(* CODESYS project Automation.library
   Company: Ziga Javornik
   DefaultNamespace: ZigaLibs.Automation
   Version: 0.0.1.2
   Placeholder: ZigaLibs.Automation
   Author: Ziga Javornik
   Description: Function blocks used for general automation.
   Title: ZigaLibs.Automation

Project tree, tasks and I/O mapping:
  libraries: Tc2_Standard, * (Beckhoff Automation GmbH); Tc2_System, * (Beckhoff Automation GmbH); Tc3_Module, * (Beckhoff Automation GmbH); TcUnit, * (www.tcunit.org); ZigaLibs.ProcessControl, 0.0.2.3 (Ziga Javornik); ZigaLibs.Core, 0.0.3.7 (Ziga Javornik)
  GVLs/
  SOURCE/
    FrequencyInverter/
      data type E_FqInverterState
      function block FB_FqInverter [ST]: CalculateFeedback, CalculateSetpoint, Enabled, Error, FB_init, Frequency, MaxFrequency, Reset, SetpointDeviation
      function block FB_FqInverter_IO [ST]: CalculateFeedback, CalculateSetpoint, Enabled, Error, FB_init, Frequency, MaxFrequency, Reset, SetpointDeviation
      interface I_FqInverter: Enabled, Error, Frequency, MaxFrequency, Reset
      data type ST_FqInverter_HwInputs
      data type ST_FqInverter_HwOutputs
    LightTower/
      function block FB_LightTower [ST]: Buzzer, FB_init, GreenLight, OrangeLight, RedLight
      function block FB_LightTowerComponent [ST]: Activate, Deactivate, FB_init, PulseWithInterval, Value
      interface I_LightTower: Buzzer, GreenLight, OrangeLight, RedLight
      interface I_LightTowerComponent: Activate, Deactivate, PulseWithInterval, Value
    MFC/
      data type ST_MfcCommands
      data type ST_MfcFeedback
  TESTS/
    Test suites/
      function block FB_FqInverter_IO_Tests [ST]: Test01_WhenDisabledOutputIsAlwaysFalse, Test02_Enable_ExpectOutputAccordingToMaxFrequencySetting, Test03_SetNegativeMaximumFrequency_ExpectOutputAlways0, Test04_SetNegativeSetpoint_ExpectOutputAlways0, Test05_DeviationIsOnlyActiveWhenEnabled, Test06_InverterErrorActive_ExpectOutputAlways0, Test07_Reset_ExpectPulseOnOutput_WhenNoErrorExpectNothing, TestXX_Template
      function block FB_LightTower_Tests [ST]: Test01_GreenLight_ActivateDeactivate_VerifyReferencedVariableValue, Test02_OrangeLight_ActivateDeactivate_VerifyReferencedVariableValue, Test03_RedLight_ActivateDeactivate_VerifyReferencedVariableValue, Test04_Buzzer_ActivateDeactivate_VerifyReferencedVariableValue
      function block FB_LightTowerComponent_Tests [ST]: Test01_AllFunctionalityTests
    program PRG_TESTS [ST]
*)

// SOURCE/FrequencyInverter/E_FqInverterState
{attribute 'qualified_only'}
{attribute 'strict'}
TYPE E_FqInverterState :
(
	DISABLED,
	ENABLED,
	RUNNING,
	ERROR,
	RESET
);
END_TYPE

// SOURCE/FrequencyInverter/ST_FqInverter_HwInputs
TYPE ST_FqInverter_HwInputs :
STRUCT
	Feedback	: INT;	// Actual feedback value
	Error		: BOOL;	// Error indication
	Ready		: BOOL;	// Ready indication
END_STRUCT
END_TYPE

// SOURCE/FrequencyInverter/ST_FqInverter_HwOutputs
TYPE ST_FqInverter_HwOutputs :
STRUCT
	Setpoint	: INT;	// Setpoint value
	Enable		: BOOL;	// Enable operation
	Reset		: BOOL;	// Reset error
END_STRUCT
END_TYPE

// SOURCE/MFC/ST_MfcCommands
TYPE ST_MfcCommands :
STRUCT
	FlowSetpoint	: REAL;
	Enable			: BOOL;
END_STRUCT
END_TYPE

// SOURCE/MFC/ST_MfcFeedback
TYPE ST_MfcFeedback :
STRUCT
	ValvePosition	: REAL;
	ActualFlow		: REAL;
END_STRUCT
END_TYPE

// SOURCE/FrequencyInverter/FB_FqInverter
// A simple frequency invert trough IO signals function block. 
// The difference to FB_FqInverter_IO is that this block uses reference assignment instead of having IO signals generated trough process image
// Constructor parameters:
(*
	(setpointMaximumValue	:= 32767,	//INT; Maximum setpoint value, ging to terminal   
	feedbackMaximumValue	:= 32767,	//INT; Maximum feedback value coming from terminal
	maximumFrequency		:= 50.0,	//REAL; Maximum frequency
	// Output signals, going to inverter
	enableSignal	:= , // REFERENCE TO BOOL;
	resetSignal		:= , // REFERENCE TO BOOL;
	setpointSignal	:= , // REFERENCE TO INT;
	// Input signals, coming from inverter
	errorSignal		:= , // REFERENCE TO BOOL;
	feedbackSignal	:= ); // REFERENCE TO INT;
*)
FUNCTION_BLOCK FB_FqInverter IMPLEMENTS I_FqInverter
VAR
	_enabled				: BOOL;
	_error					: BOOL;
	_frequency				: ZigaLibs_Core.ST_Value;
	_maxFrequency			: REAL;
	_state					: E_FqInverterState;
	_setpointMaximumValue	: INT;
	_feedbackMaximumValue	: INT;
	_setpointDeviation			: ZigaLibs_ProcessControl.FB_ValueDeviation;
	
	// Output signals, going to inverter
	_enableSignal	: REFERENCE TO BOOL;
	_resetSignal	: REFERENCE TO BOOL;
	_setpointSignal	: REFERENCE TO INT;
	// Input signals, coming from inverter
	_errorSignal	: REFERENCE TO BOOL;
	_feedbackSignal	: REFERENCE TO INT;
END_VAR

_frequency.Actual := CalculateFeedback();

IF _errorSignal AND _state <> E_FqInverterState.RESET THEN
	_State := E_FqInverterState.ERROR;
END_IF


CASE _state OF
	E_FqInverterState.DISABLED:
		_enableSignal := FALSE;
		_setpointSignal := 0;
		IF _enabled THEN
			_state := E_FqInverterState.ENABLED;
		END_IF
		
	E_FqInverterState.ENABLED:
		IF NOT _enabled THEN
			_state := E_FqInverterState.DISABLED;
		ELSE
			_enableSignal := TRUE;
			_setpointSignal := CalculateSetpoint();
		END_IF
		
	E_FqInverterState.ERROR:
		_error := TRUE;
		_enableSignal := FALSE;
		_setpointSignal := 0;
		
	E_FqInverterState.RESET:
		_error := FALSE;
		_enableSignal := FALSE;
		_setpointSignal := 0;
		_resetSignal := FALSE;
		IF NOT _errorSignal THEN
			_state := E_FqInverterState.DISABLED;
		END_IF
END_CASE

_setpointDeviation.Enable := _state = E_FqInverterState.ENABLED;
_setpointDeviation.Value.Actual := _frequency.Actual;
_setpointDeviation.Value.Setpoint := _frequency.Setpoint;
_setpointDeviation();

METHOD PRIVATE CalculateFeedback : REAL
VAR_INPUT
END_VAR
// Invalid parameter setting.
IF _feedbackMaximumValue <= 0 OR _maxFrequency < 0 THEN
	CalculateFeedback := 0;
ELSE
	CalculateFeedback := _maxFrequency * (INT_TO_REAL(_feedbackSignal) / INT_TO_REAL(_feedbackMaximumValue));
END_IF
END_METHOD

METHOD PRIVATE CalculateSetpoint : INT
VAR_INPUT
END_VAR
VAR
	validatedFrequencySetpoint	: REAL;
	frequencySetpointFraction	: REAL;
END_VAR
// Limit setpoint between 0 and max
validatedFrequencySetpoint := MAX(0, MIN(_maxFrequency, _frequency.Setpoint));

// If max frequency is 0, invalid setting
IF _maxFrequency <= 0 THEN
	frequencySetpointFraction := 0;
ELSE
	frequencySetpointFraction := validatedFrequencySetpoint / _maxFrequency;
END_IF

CalculateSetpoint := REAL_TO_INT(frequencySetpointFraction * _setpointMaximumValue);
END_METHOD

{attribute 'monitoring':='call'}
(* Gets or sets whether or not the unit is enabled.*)
PROPERTY Enabled : BOOL
GET
Enabled := _enabled;
END_GET
SET
_enabled := Enabled;
END_SET
END_PROPERTY

{attribute 'monitoring':='call'}
(* Returns TRUE if an error is active*)
PROPERTY Error : BOOL
GET
Error := _error;
END_GET
END_PROPERTY

METHOD FB_init : BOOL
VAR_INPUT
	bInitRetains : BOOL; // if TRUE, the retain variables are initialized (warm start / cold start)
	bInCopyCode : BOOL;  // if TRUE, the instance afterwards gets moved into the copy code (online change)
	setpointMaximumValue	: INT;	// Maximum setpoint value, ging to terminal
	feedbackMaximumValue	: INT;	// Maximum feedback value coming from terminal
	maximumFrequency		: REAL;	// Maximum frequency
	// Output signals, going to inverter
	enableSignal	: REFERENCE TO BOOL;
	resetSignal		: REFERENCE TO BOOL;
	setpointSignal	: REFERENCE TO INT;
	// Input signals, coming from inverter
	errorSignal		: REFERENCE TO BOOL;
	feedbackSignal	: REFERENCE TO INT;
END_VAR
_setpointMaximumValue := setpointMaximumValue;
_feedbackMaximumValue := feedbackMaximumValue;
_maxFrequency := maximumFrequency;
_enableSignal REF= enableSignal;
_resetSignal REF= resetSignal;
_setpointSignal REF= setpointSignal;
_errorSignal REF= errorSignal;
_feedbackSignal REF= feedbackSignal;
END_METHOD

{attribute 'monitoring':='call'}
(* Provides access to frequncy setpoint and actual value*)
PROPERTY Frequency : REFERENCE TO ZigaLibs_Core.ST_Value
GET
Frequency REF= _frequency;
END_GET
SET
_frequency := Frequency;
END_SET
END_PROPERTY

{attribute 'monitoring':='call'}
(* Gets or sets the maximum frequency.*)
PROPERTY MaxFrequency : REAL
GET
MaxFrequency := _maxFrequency;
END_GET
SET
_maxFrequency := MaxFrequency;
END_SET
END_PROPERTY

(* If an error is active, it will be reset.*)
METHOD Reset
VAR_INST
	resetTimer	: Tc2_Standard.TON := (PT := T#200MS);
END_VAR
IF _errorSignal THEN
	resetTimer(IN := NOT resetTimer.Q, PT := T#100MS);
	_resetSignal := NOT resetTimer.Q;
ELSE
	resetTimer(IN := FALSE);
	_resetSignal := FALSE;
	_state := E_FqInverterState.RESET;
END_IF
END_METHOD

{attribute 'monitoring':='call'}
PROPERTY SetpointDeviation : ZigaLibs_ProcessControl.I_ValueDeviationLimited
GET
SetpointDeviation := _setpointDeviation;
END_GET
END_PROPERTY

END_FUNCTION_BLOCK

// SOURCE/FrequencyInverter/FB_FqInverter_IO
// A simple frequency invert trough IO signals function block
// Constructor parameters:
(*
	(setpointMaximumValue	:= 32767,	//INT; Maximum setpoint value, ging to terminal   
	feedbackMaximumValue	:= 32767,	//INT; Maximum feedback value coming from terminal
	maximumFrequency		:= 50.0);	//REAL; Maximum frequency                         

*)
FUNCTION_BLOCK FB_FqInverter_IO IMPLEMENTS I_FqInverter
VAR
	_enabled				: BOOL;
	_error					: BOOL;
	_frequency				: ZigaLibs_Core.ST_Value;
	_maxFrequency			: REAL;
	_state					: E_FqInverterState;
	_setpointMaximumValue	: INT;
	_feedbackMaximumValue	: INT;
	_setpointDeviation			: ZigaLibs_ProcessControl.FB_ValueDeviation;
END_VAR

VAR
	Inputs	AT %I* 	: ST_FqInverter_HwInputs;
	Outputs	AT %Q*	: ST_FqInverter_HwOutputs;
END_VAR

_frequency.Actual := CalculateFeedback();

IF Inputs.Error AND _state <> E_FqInverterState.RESET THEN
	_State := E_FqInverterState.ERROR;
END_IF


CASE _state OF
	E_FqInverterState.DISABLED:
		Outputs.Enable := FALSE;
		Outputs.Setpoint := 0;
		IF _enabled THEN
			_state := E_FqInverterState.ENABLED;
		END_IF
		
	E_FqInverterState.ENABLED:
		IF NOT _enabled THEN
			_state := E_FqInverterState.DISABLED;
		ELSE
			Outputs.Enable := TRUE;
			Outputs.Setpoint := CalculateSetpoint();
		END_IF
		
	E_FqInverterState.ERROR:
		_error := TRUE;
		Outputs.Enable := FALSE;
		Outputs.Setpoint := 0;
		
	E_FqInverterState.RESET:
		_error := FALSE;
		Outputs.Enable := FALSE;
		Outputs.Setpoint := 0;
		outputs.Reset := FALSE;
		IF NOT Inputs.Error THEN
			_state := E_FqInverterState.DISABLED;
		END_IF
END_CASE

_setpointDeviation.Enable := _state = E_FqInverterState.ENABLED;
_setpointDeviation.Value.Actual := _frequency.Actual;
_setpointDeviation.Value.Setpoint := _frequency.Setpoint;
_setpointDeviation();

METHOD PRIVATE CalculateFeedback : REAL
VAR_INPUT
END_VAR
// Invalid parameter setting.
IF _feedbackMaximumValue <= 0 OR _maxFrequency < 0 THEN
	CalculateFeedback := 0;
ELSE
	CalculateFeedback := _maxFrequency * (INT_TO_REAL(Inputs.Feedback) / INT_TO_REAL(_feedbackMaximumValue));
END_IF
END_METHOD

METHOD PRIVATE CalculateSetpoint : INT
VAR_INPUT
END_VAR
VAR
	validatedFrequencySetpoint	: REAL;
	frequencySetpointFraction	: REAL;
END_VAR
// Limit setpoint between 0 and max
validatedFrequencySetpoint := MAX(0, MIN(_maxFrequency, _frequency.Setpoint));

// If max frequency is 0, invalid setting
IF _maxFrequency <= 0 THEN
	frequencySetpointFraction := 0;
ELSE
	frequencySetpointFraction := validatedFrequencySetpoint / _maxFrequency;
END_IF

CalculateSetpoint := REAL_TO_INT(frequencySetpointFraction * _setpointMaximumValue);
END_METHOD

{attribute 'monitoring':='call'}
(* Gets or sets whether or not the unit is enabled.*)
PROPERTY Enabled : BOOL
GET
Enabled := _enabled;
END_GET
SET
_enabled := Enabled;
END_SET
END_PROPERTY

{attribute 'monitoring':='call'}
(* Returns TRUE if an error is active*)
PROPERTY Error : BOOL
GET
Error := _error;
END_GET
END_PROPERTY

METHOD FB_init : BOOL
VAR_INPUT
	bInitRetains : BOOL; // if TRUE, the retain variables are initialized (warm start / cold start)
	bInCopyCode : BOOL;  // if TRUE, the instance afterwards gets moved into the copy code (online change)
	setpointMaximumValue	: INT;	// Maximum setpoint value, ging to terminal
	feedbackMaximumValue	: INT;	// Maximum feedback value coming from terminal
	maximumFrequency		: REAL;	// Maximum frequency
END_VAR
_setpointMaximumValue := setpointMaximumValue;
_feedbackMaximumValue := feedbackMaximumValue;
_maxFrequency := maximumFrequency;
END_METHOD

{attribute 'monitoring':='call'}
(* Provides access to frequncy setpoint and actual value*)
PROPERTY Frequency : REFERENCE TO ZigaLibs_Core.ST_Value
GET
Frequency REF= _frequency;
END_GET
SET
_frequency := Frequency;
END_SET
END_PROPERTY

{attribute 'monitoring':='call'}
(* Gets or sets the maximum frequency.*)
PROPERTY MaxFrequency : REAL
GET
MaxFrequency := _maxFrequency;
END_GET
SET
_maxFrequency := MaxFrequency;
END_SET
END_PROPERTY

(* If an error is active, it will be reset.*)
METHOD Reset
VAR_INST
	resetTimer	: Tc2_Standard.TON := (PT := T#200MS);
END_VAR
IF Inputs.Error THEN
	resetTimer(IN := NOT resetTimer.Q, PT := T#100MS);
	Outputs.Reset := NOT resetTimer.Q;
ELSE
	resetTimer(IN := FALSE);
	Outputs.Reset := FALSE;
	_state := E_FqInverterState.RESET;
END_IF
END_METHOD

{attribute 'monitoring':='call'}
PROPERTY SetpointDeviation : ZigaLibs_ProcessControl.I_ValueDeviationLimited
GET
SetpointDeviation := _setpointDeviation;
END_GET
END_PROPERTY

END_FUNCTION_BLOCK

// SOURCE/FrequencyInverter/I_FqInverter
INTERFACE I_FqInverter

{attribute 'monitoring':='call'}
// Gets or sets whether or not the unit is enabled.
PROPERTY Enabled : BOOL
GET
END_GET
SET
END_SET
END_PROPERTY

{attribute 'monitoring':='call'}
// Returns TRUE if an error is active
PROPERTY Error : BOOL
GET
END_GET
END_PROPERTY

{attribute 'monitoring':='call'}
// Provides access to frequncy setpoint and actual value
PROPERTY Frequency : REFERENCE TO ZigaLibs_Core.ST_Value
GET
END_GET
SET
END_SET
END_PROPERTY

{attribute 'monitoring':='call'}
// Gets or sets the maximum frequency.
PROPERTY MaxFrequency : REAL
GET
END_GET
SET
END_SET
END_PROPERTY

// If an error is active, it will be reset.
METHOD Reset
END_METHOD

END_INTERFACE

// SOURCE/LightTower/FB_LightTower
(* Provides acces to control the light tower components.
Constructor template as follows:
	(greenLight		:= ,// REFERENCE TO BOOL;
	orangeLight		:= ,// REFERENCE TO BOOL;
	redLight		:= ,// REFERENCE TO BOOL;
	buzzer			:= );// REFERENCE TO BOOL;
*)

FUNCTION_BLOCK FB_LightTower IMPLEMENTS I_LightTower
VAR	
	_redLightControl	: FB_LightTowerComponent;
	_orangeLightControl	: FB_LightTowerComponent;
	_greenLightControl	: FB_LightTowerComponent;
	_buzzerControl		: FB_LightTowerComponent;
END_VAR

_redLightControl();
_orangeLightControl();
_greenLightControl();
_buzzerControl();

// Provides access to buzzer control
PROPERTY Buzzer : I_LightTowerComponent
GET
Buzzer := _buzzerControl;
END_GET
END_PROPERTY

METHOD FB_init : BOOL
VAR_INPUT
	bInitRetains 	: BOOL; // if TRUE, the retain variables are initialized (warm start / cold start)
	bInCopyCode 	: BOOL;  // if TRUE, the instance afterwards gets moved into the copy code (online change)
	greenLight		: REFERENCE TO BOOL;
	orangeLight		: REFERENCE TO BOOL;
	redLight		: REFERENCE TO BOOL;
	buzzer			: REFERENCE TO BOOL;
END_VAR
_greenLightControl.component REF= greenLight;
_orangeLightControl.component REF= orangeLight;
_redLightControl.component REF= redLight;
_buzzerControl.component REF= buzzer;
END_METHOD

// Provides access to green light control
PROPERTY GreenLight : I_LightTowerComponent
GET
GreenLight := _greenLightControl;
END_GET
END_PROPERTY

// Provides access to orange light control
PROPERTY OrangeLight : I_LightTowerComponent
GET
OrangeLight := _orangeLightControl;
END_GET
END_PROPERTY

// Provides access to red light control
PROPERTY RedLight : I_LightTowerComponent
GET
RedLight := _redLightControl;
END_GET
END_PROPERTY

END_FUNCTION_BLOCK

// SOURCE/LightTower/I_LightTower
INTERFACE I_LightTower

// Provides access to buzzer control
PROPERTY Buzzer : I_LightTowerComponent
GET
END_GET
END_PROPERTY

// Provides access to green light control
PROPERTY GreenLight : I_LightTowerComponent
GET
END_GET
END_PROPERTY

// Provides access to orange light control
PROPERTY OrangeLight : I_LightTowerComponent
GET
END_GET
END_PROPERTY

// Provides access to red light control
PROPERTY RedLight : I_LightTowerComponent
GET
END_GET
END_PROPERTY

END_INTERFACE

// SOURCE/LightTower/I_LightTowerComponent
INTERFACE I_LightTowerComponent

// Sets the component state to TRUE.
METHOD Activate
VAR_INPUT
END_VAR
END_METHOD

// Sets the component state to FALSE.
METHOD Deactivate
VAR_INPUT
END_VAR
END_METHOD

METHOD PulseWithInterval
VAR_INPUT
	DurationOn	: TIME;
	DurationOff	: TIME;
END_VAR
END_METHOD

{attribute 'monitoring':='call'}
// Gets the current state of the component
PROPERTY Value : BOOL
GET
END_GET
END_PROPERTY

END_INTERFACE

// SOURCE/LightTower/FB_LightTowerComponent
FUNCTION_BLOCK FB_LightTowerComponent IMPLEMENTS I_LightTowerComponent
VAR_INPUT
	component : REFERENCE TO BOOL;
END_VAR
VAR
	_component	: ZigaLibs_Core.BoolEx := (variable := component);
END_VAR

_component(variable := component);

METHOD Activate
IF NOT __ISVALIDREF(component) THEN
	RETURN;
END_IF
_component.Set();
END_METHOD

METHOD Deactivate
IF NOT __ISVALIDREF(component) THEN
	RETURN;
END_IF
_component.Reset();
END_METHOD

METHOD FB_init : BOOL
VAR_INPUT
	bInitRetains : BOOL; // if TRUE, the retain variables are initialized (warm start / cold start)
	bInCopyCode : BOOL;  // if TRUE, the instance afterwards gets moved into the copy code (online change)
END_VAR
END_METHOD

METHOD PulseWithInterval
VAR_INPUT
	DurationOn	: TIME;
	DurationOff	: TIME;
END_VAR
VAR_INST
	timerOn		: Tc2_Standard.TON;
	timerOff	: Tc2_Standard.TON;
END_VAR
IF NOT __ISVALIDREF(component) THEN
	RETURN;
END_IF
_component.PulseWithInterval(DurationOn,DurationOff);
END_METHOD

{attribute 'monitoring':='call'}
(* Gets the current state of the component*)
PROPERTY Value : BOOL
GET
Value := _component.Value;
END_GET
END_PROPERTY

END_FUNCTION_BLOCK

// TESTS/Test suites/FB_FqInverter_IO_Tests
FUNCTION_BLOCK INTERNAL FB_FqInverter_IO_Tests EXTENDS FB_TestSuite
VAR_INPUT
END_VAR
VAR_OUTPUT
END_VAR
VAR
	_fqInvert : FB_FqInverter_IO(
		setpointMaximumValue	:= 32767,	//INT; Maximum setpoint value, ging to terminal   
		feedbackMaximumValue	:= 32767,	//INT; Maximum feedback value coming from terminal
		maximumFrequency		:= 50.0);	//REAL; Maximum frequency     
END_VAR

Test01_WhenDisabledOutputIsAlwaysFalse();
Test02_Enable_ExpectOutputAccordingToMaxFrequencySetting();
Test03_SetNegativeMaximumFrequency_ExpectOutputAlways0();
Test04_SetNegativeSetpoint_ExpectOutputAlways0();
Test05_DeviationIsOnlyActiveWhenEnabled();
Test06_InverterErrorActive_ExpectOutputAlways0();
Test07_Reset_ExpectPulseOnOutput_WhenNoErrorExpectNothing();

METHOD Test01_WhenDisabledOutputIsAlwaysFalse
VAR_INPUT
END_VAR
IF TcUnit.TEST_ORDERED('Test01_WhenDisabledOutputIsAlwaysFalse') THEN
	_fqInvert.Enabled := FALSE;
	_fqInvert.Frequency.Setpoint := 0;
	AssertEquals_INT(
		Actual := _fqInvert.Outputs.Setpoint,
		Expected := 0,
		Message := 'When disabled and setpoint is 0, expected output is also 0.');
		
	_fqInvert.Frequency.Setpoint := 100;
	AssertEquals_INT(
		Actual := _fqInvert.Outputs.Setpoint,
		Expected := 0,
		Message := 'When disabled and setpoint is 50, expected output is also 0.');
	TcUnit.TEST_FINISHED();
END_IF
END_METHOD

METHOD Test02_Enable_ExpectOutputAccordingToMaxFrequencySetting
VAR_INPUT
END_VAR
IF TcUnit.TEST_ORDERED('Test02_Enable_ExpectOutputAccordingToMaxFrequencySetting') THEN
	_fqInvert.Enabled := TRUE;
	_fqInvert.Frequency.Setpoint := 0;
	_fqInvert();
	AssertEquals_INT(
		Actual := _fqInvert.Outputs.Setpoint,
		Expected := 0,
		Message := 'When enabled and setpoint is 0, expected output is also 0.');

	
	_fqInvert.Frequency.Setpoint := 10;
	_fqInvert();
	AssertEquals_INT(
		Actual := _fqInvert.Outputs.Setpoint,
		Expected := 6553,
		Message := 'When enabled, max fq 50 and setpoint is 10, expected output is also 20% of 32767.');
		
	TcUnit.WRITE_PROTECTED_INT(
		Ptr := ADR(_fqInvert.Inputs.Feedback),
	 	Value := _fqInvert.Outputs.Setpoint);
	_fqInvert();
	AssertEquals_REAL(
		Actual := _fqInvert.Frequency.Actual,
		Expected := _fqInvert.Frequency.Setpoint,
		Delta := 0.001,
		Message := 'Setpoint and feedback should be the same (test sets input value to same as output) - scaling incorrect');
		
	_fqInvert.Frequency.Setpoint := 50;
	_fqInvert();
	AssertEquals_INT(
		Actual := _fqInvert.Outputs.Setpoint,
		Expected := 32767,
		Message := 'When enabled, max fq 50 and setpoint is 50, expected output is 32767.');
		
	_fqInvert.Frequency.Setpoint := 100;
	_fqInvert();
	AssertEquals_INT(
		Actual := _fqInvert.Outputs.Setpoint,
		Expected := 32767,
		Message := 'When enabled, max fq 50 and setpoint is 100, expected output is 32767.');
		
	TcUnit.WRITE_PROTECTED_INT(
		Ptr := ADR(_fqInvert.Inputs.Feedback),
	 	Value := _fqInvert.Outputs.Setpoint);	
	_fqInvert();
	AssertEquals_REAL(
		Actual := _fqInvert.Frequency.Actual,
		Expected := 50.0,
		Delta := 0.001,
		Message := 'When setting frequency to 100 and max is 50, expected actual frequency is 50 (test sets input)');
		
	TcUnit.TEST_FINISHED();
END_IF
END_METHOD

METHOD Test03_SetNegativeMaximumFrequency_ExpectOutputAlways0
VAR_INPUT
END_VAR
IF TcUnit.TEST_ORDERED('Test03_SetNegativeMaximumFrequency_ExpectOutputAlways0') THEN
	_fqInvert.MaxFrequency := -50;
	_fqInvert.Frequency.Setpoint := 50;
	_fqInvert.Enabled := TRUE;
	_fqInvert();
	AssertEquals_INT(
		Actual := _fqInvert.Outputs.Setpoint,
		Expected := 0,
		Message := 'Negative maximum frequency should be treated as an error, no output should be generated.');
	
	_fqInvert.Enabled := FALSE;
	_fqInvert();
	AssertEquals_INT(
		Actual := _fqInvert.Outputs.Setpoint,
		Expected := 0,
		Message := 'Negative maximum frequency while disabled should be treated as an error, no output should be generated.');
		
	_fqInvert.Enabled := TRUE;	
	_fqInvert.MaxFrequency := -300;
	_fqInvert();
	AssertEquals_INT(
		Actual := _fqInvert.Outputs.Setpoint,
		Expected := 0,
		Message := 'Negative maximum frequency should be treated as an error, no output should be generated.');
	TcUnit.TEST_FINISHED();
END_IF
END_METHOD

METHOD Test04_SetNegativeSetpoint_ExpectOutputAlways0
VAR_INPUT
END_VAR
IF TcUnit.TEST_ORDERED('Test04_SetNegativeSetpoint_ExpectOutputAlways0') THEN
	_fqInvert.MaxFrequency := 100;
	_fqInvert.Frequency.Setpoint := -100;
	_fqInvert.Enabled := TRUE;
	_fqInvert();
	AssertEquals_INT(
		Actual := _fqInvert.Outputs.Setpoint,
		Expected := 0,
		Message := 'Negative setpoint should be treated as an error, no output should be generated.');
	TcUnit.TEST_FINISHED();
END_IF
END_METHOD

METHOD Test05_DeviationIsOnlyActiveWhenEnabled
VAR_INPUT
END_VAR
IF TcUnit.TEST_ORDERED('Test05_DeviationIsOnlyActiveWhenEnabled') THEN
	TcUnit.WRITE_PROTECTED_INT(Ptr := ADR(_fqInvert.Inputs.Feedback), 0);
	_fqInvert.Enabled := FALSE;
	_fqInvert.SetpointDeviation.ActivationDelay := T#0S;
	_fqInvert.SetpointDeviation.MaxDeviation := 0;
	_fqInvert.Frequency.Setpoint := 50;
	_fqInvert();
	AssertTrue(
		Condition := _fqInvert.SetpointDeviation.Status = ZigaLibs_ProcessControl.E_ValueDeviationStatus.OK,
		Message := 'When inverter is disabled, setpoint deviation should be inactive and should report OK.');
		
	_fqInvert.Enabled := TRUE;
	_fqInvert();
	AssertTrue(
		Condition := _fqInvert.SetpointDeviation.Status = ZigaLibs_ProcessControl.E_ValueDeviationStatus.NOK,
		Message := 'When inverter is enabled, setpoint deviation should be active and should report NOK if deviation is active.');
	
	_fqInvert.Frequency.Setpoint := 0;	
	_fqInvert();
	AssertTrue(
		Condition := _fqInvert.SetpointDeviation.Status = ZigaLibs_ProcessControl.E_ValueDeviationStatus.OK,
		Message := 'When inverter is enabled, if there is no deviation, status should be OK.');
	
	_fqInvert.SetpointDeviation.MaxDeviation := 0.01; 
	_fqInvert.Frequency.Setpoint := 0.02;	
	_fqInvert();
	AssertTrue(
		Condition := _fqInvert.SetpointDeviation.Status = ZigaLibs_ProcessControl.E_ValueDeviationStatus.NOK,
		Message := 'When inverter is enabled, if there is deviation, status should be NOK.');
		
	_fqInvert.Enabled := FALSE;
	_fqInvert();
	AssertTrue(
		Condition := _fqInvert.SetpointDeviation.Status = ZigaLibs_ProcessControl.E_ValueDeviationStatus.OK,
		Message := 'When inverter is disabled, if there was deviation, it should be cleared since inverter is disabled.');
		
	TcUnit.TEST_FINISHED();
END_IF
END_METHOD

METHOD Test06_InverterErrorActive_ExpectOutputAlways0
VAR_INPUT
END_VAR
IF TcUnit.TEST_ORDERED('Test06_InverterErrorActive_ExpectOutputAlways0') THEN
	TcUnit.WRITE_PROTECTED_BOOL(Ptr := ADR(_fqInvert.Inputs.Error), TRUE);
	_fqInvert.Frequency.Setpoint := 50;
	_fqInvert.Enabled := FALSE;
	_fqInvert();
	AssertEquals_INT(
		Actual := _fqInvert.Outputs.Setpoint,
		Expected := 0,
		Message := 'If an error is active and disabled, output should always be 0.');
		
	_fqInvert.Enabled := TRUE;
	_fqInvert();
	AssertEquals_INT(
		Actual := _fqInvert.Outputs.Setpoint,
		Expected := 0,
		Message := 'If an error is active and enabled, output should always be 0.');
		
	TcUnit.WRITE_PROTECTED_BOOL(Ptr := ADR(_fqInvert.Inputs.Error), FALSE);	
	TcUnit.TEST_FINISHED();
END_IF
END_METHOD

METHOD Test07_Reset_ExpectPulseOnOutput_WhenNoErrorExpectNothing
VAR_INPUT
END_VAR
IF TcUnit.TEST_ORDERED('Test07_Reset_ExpectPulseOnOutput_WhenNoErrorExpectNothing') THEN
	TcUnit.WRITE_PROTECTED_BOOL(Ptr := ADR(_fqInvert.Inputs.Error), Value := TRUE);
	_fqInvert.Reset();
	_fqInvert();
	AssertTrue(
		Condition := _fqInvert.Outputs.Reset,
		Message := 'If an error is active, calling .Reset() should generate a pulse');		
	
	TcUnit.WRITE_PROTECTED_BOOL(Ptr := ADR(_fqInvert.Inputs.Error), Value := FALSE);
	_fqInvert.Reset();
	_fqInvert();
	AssertFalse(
		Condition := _fqInvert.Outputs.Reset,
		Message := 'If an error is not active, calling .Reset() should not generate a pulse');
		
	TcUnit.TEST_FINISHED();
END_IF
END_METHOD

METHOD TestXX_Template
VAR_INPUT
END_VAR
IF TcUnit.TEST_ORDERED('TestXX_Template') THEN
	
	TcUnit.TEST_FINISHED();
END_IF
END_METHOD

END_FUNCTION_BLOCK

// TESTS/Test suites/FB_LightTower_Tests
FUNCTION_BLOCK INTERNAL FB_LightTower_Tests EXTENDS FB_TestSuite
VAR_INPUT
END_VAR
VAR_OUTPUT
END_VAR
VAR
	redLight	: BOOL;
	greenLight	: BOOL;
	orangeLight	: BOOL;
	buzzer		: BOOL;
	lightTower	: FB_LightTower	(
		greenLight		:= greenLight,// REFERENCE TO BOOL;
		orangeLight		:= orangeLight ,// REFERENCE TO BOOL;
		redLight		:= redLight,// REFERENCE TO BOOL;
		buzzer			:= buzzer);// REFERENCE TO BOOL;

END_VAR

lightTower();

Test01_GreenLight_ActivateDeactivate_VerifyReferencedVariableValue();
Test02_OrangeLight_ActivateDeactivate_VerifyReferencedVariableValue();
Test03_RedLight_ActivateDeactivate_VerifyReferencedVariableValue();
Test04_Buzzer_ActivateDeactivate_VerifyReferencedVariableValue();

METHOD PRIVATE Test01_GreenLight_ActivateDeactivate_VerifyReferencedVariableValue
VAR_INPUT
END_VAR
IF TcUnit.TEST_ORDERED('Test01_GreenLight_ActivateDeactivate_VerifyReferencedVariableValue') THEN
	lightTower.GreenLight.Activate();
	AssertTrue(Condition := greenLight, Message := 'Activating green light failed');
	AssertFalse(Condition := orangeLight, Message := 'Activating green light should not affect orange light.');
	AssertFalse(Condition := redLight, Message := 'Activating green light should not affect red light.');	
	AssertFalse(Condition := buzzer, Message := 'Activating green light should not affect buzzer.');
		
	lightTower.GreenLight.Deactivate();
	AssertFalse(Condition := greenLight, Message := 'Deactivating green light failed');
	AssertFalse(Condition := orangeLight, Message := 'Deactivating green light should not affect orange light.');
	AssertFalse(Condition := redLight, Message := 'Deactivating green light should not affect red light.');	
	AssertFalse(Condition := buzzer, Message := 'Deactivating green light should not affect buzzer.');
	
	TcUnit.TEST_FINISHED();
END_IF
END_METHOD

METHOD PRIVATE Test02_OrangeLight_ActivateDeactivate_VerifyReferencedVariableValue
VAR_INPUT
END_VAR
IF TcUnit.TEST_ORDERED('Test02_OrangeLight_ActivateDeactivate_VerifyReferencedVariableValue') THEN
	lightTower.OrangeLight.Activate();
	AssertTrue(Condition := orangeLight, Message := 'Activating orange light failed');
	AssertFalse(Condition := greenLight, Message := 'Activating orange light should not affect green light.');
	AssertFalse(Condition := redLight, Message := 'Activating orange light should not affect red light.');	
	AssertFalse(Condition := buzzer, Message := 'Activating orange light should not affect buzzer.');
		
	lightTower.OrangeLight.Deactivate();
	AssertFalse(Condition := orangeLight, Message := 'Deactivating orange light failed');
	AssertFalse(Condition := greenLight, Message := 'Deactivating orange light should not affect green light.');
	AssertFalse(Condition := redLight, Message := 'Deactivating orange light should not affect red light.');	
	AssertFalse(Condition := buzzer, Message := 'Deactivating orange light should not affect buzzer.');
	
	TcUnit.TEST_FINISHED();
END_IF
END_METHOD

METHOD PRIVATE Test03_RedLight_ActivateDeactivate_VerifyReferencedVariableValue
VAR_INPUT
END_VAR
IF TcUnit.TEST_ORDERED('Test03_RedLight_ActivateDeactivate_VerifyReferencedVariableValue') THEN
	lightTower.RedLight.Activate();
	AssertTrue(Condition := redLight, Message := 'Activating red light failed');
	AssertFalse(Condition := greenLight, Message := 'Activating red light should not affect green light.');
	AssertFalse(Condition := orangeLight, Message := 'Activating red light should not affect orange light.');	
	AssertFalse(Condition := buzzer, Message := 'Activating red light should not affect buzzer.');
		
	lightTower.RedLight.Deactivate();
	AssertFalse(Condition := redLight, Message := 'Deactivating red light failed');
	AssertFalse(Condition := greenLight, Message := 'Deactivating red light should not affect green light.');
	AssertFalse(Condition := orangeLight, Message := 'Deactivating red light should not affect orange light.');	
	AssertFalse(Condition := buzzer, Message := 'Deactivating red light should not affect buzzer.');
	
	TcUnit.TEST_FINISHED();
END_IF
END_METHOD

METHOD PRIVATE Test04_Buzzer_ActivateDeactivate_VerifyReferencedVariableValue
VAR_INPUT
END_VAR
IF TcUnit.TEST_ORDERED('Test04_Buzzer_ActivateDeactivate_VerifyReferencedVariableValue') THEN
	lightTower.Buzzer.Activate();
	AssertTrue(Condition := buzzer, Message := 'Activating buzzer failed');
	AssertFalse(Condition := greenLight, Message := 'Activating buzzer should not affect green light.');
	AssertFalse(Condition := orangeLight, Message := 'Activating buzzer should not affect orange light.');	
	AssertFalse(Condition := redLight, Message := 'Activating buzzer should not affect red light.');
		
	lightTower.Buzzer.Deactivate();
	AssertFalse(Condition := buzzer, Message := 'Deactivating buzzer light failed');
	AssertFalse(Condition := greenLight, Message := 'Deactivating buzzer should not affect green light.');
	AssertFalse(Condition := orangeLight, Message := 'Deactivating buzzer should not affect orange light.');	
	AssertFalse(Condition := redLight, Message := 'Deactivating buzzer should not affect red light.');
	
	TcUnit.TEST_FINISHED();
END_IF
END_METHOD

END_FUNCTION_BLOCK

// TESTS/Test suites/FB_LightTowerComponent_Tests
FUNCTION_BLOCK INTERNAL FB_LightTowerComponent_Tests EXTENDS FB_TestSuite
VAR_INPUT
END_VAR
VAR_OUTPUT
END_VAR
VAR
	componentItem	: BOOL;
END_VAR

Test01_AllFunctionalityTests();

METHOD Test01_AllFunctionalityTests 
VAR_INST
	timer	 		: Tc2_Standard.TON;
	timerOff		: Tc2_Standard.TON;
	component		: FB_LightTowerComponent := (component := componentItem);
	onOffTestDone	: BOOL;
END_VAR
IF TcUnit.TEST_ORDERED('Test01_AllFunctionalityTests') THEN
	component();
	IF NOT onOffTestDone THEN
		component.Activate();
		AssertTrue(Condition := component.Value, Message := 'Calling .Activate() should set the .Value property to TRUE.');
		AssertTrue(Condition := componentItem, Message := 'Calling .Activate() should set the referenced variable to TRUE.');
		component.Deactivate();
		AssertFalse(Condition := component.Value, Message := 'Calling .Deactivate() should set the .Value property to FALSE.');
		AssertFalse(Condition := componentItem, Message := 'Calling .Deactivate() should set the referenced variable to FALSE.');
		onOffTestDone := TRUE;
	END_IF
	
	component.PulseWithInterval(DurationOn := T#100MS, DurationOff := T#100MS);
	timer(in := TRUE, PT := T#100MS);
	IF NOT timer.Q THEN
		AssertTrue(Condition := component.Value, Message := 'Component.Value should be TRUE until duration on is elapsed.');
		AssertTrue(Condition := componentItem, Message := 'Referenced variable should be TRUE until duration on is elapsed.');
	ELSE
		timerOff(IN := TRUE, PT := T#100MS);
		IF timerOff.Q THEN
			AssertTrue(Condition := component.Value, Message := 'Component.Value should be TRUE when duration off is elapsed.');
			AssertTrue(Condition := componentItem, Message := 'Reference variable should be TRUE when duration off is elapsed.');
			TcUnit.TEST_FINISHED();
			RETURN;
		END_IF
		AssertFalse(Condition := component.Value, Message := 'Component.Value should be FALSE until duration off is elapsed.');
		AssertFalse(Condition := componentItem, Message := 'Reference variable should be FALSE until duration off is elapsed.');
	END_IF	
END_IF
END_METHOD

END_FUNCTION_BLOCK

// TESTS/PRG_TESTS
PROGRAM INTERNAL PRG_TESTS

(* Instantiate test suites here. Naming convention for tests should be a suffix with _Tests.
Good practice for creating test methods is to end them with _test as well. *)
VAR
	LightTowerComponentTest	: FB_LightTowerComponent_Tests;
	FqInverter_IOTests		: FB_FqInverter_IO_Tests;
	LighttowerTests			: FB_LightTower_Tests;
END_VAR

// Run tests in paralel
//TcUnit.RUN();

// Run tests in sequence, one after the other. Uncomment if required.
TcUnit.RUN_IN_SEQUENCE();

END_PROGRAM
